TYPE E_AlarmLevel : (
    ALARM_LEVEL_NONE := 0,
    ALARM_LEVEL_WARNING := 10,
    ALARM_LEVEL_NOK := 20,
    ALARM_LEVEL_FAULT := 30
); END_TYPE

(* stored: Version 1.1.0.1
   DUT E_AlarmLevel: Id {E3000000-0000-4000-8000-000000000015} *)
